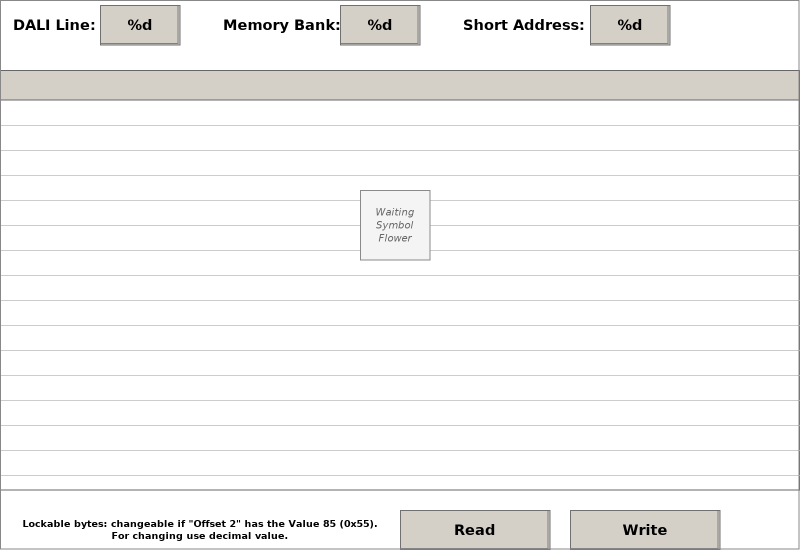
VISUALIZATION Visu_Part102MemoryBank  // 800x550
    Table (0,70 800x420), data array: DALI_Commissioning.fbPart102MemoryPages.aMemoryBank
        p1137915858: DALI_Commissioning.fbPart102MemoryPages.nOffset
        p3854506369: DALI_Commissioning.fbPart102MemoryPages.aMemoryBank[INDEX].sOffset
        p1892666644: DALI_Commissioning.fbPart102MemoryPages.aMemoryBank[INDEX].sName
        p338671338: DALI_Commissioning.fbPart102MemoryPages.aMemoryBank[INDEX].nValueDec
        p2170511999: DALI_Commissioning.fbPart102MemoryPages.aMemoryBank[INDEX].nValueHex
        p1755163831: Value Dec
        p4092479075: Value Hex
        Columns.Column.[0].Template: DALI_Commissioning.fbPart102MemoryPages.aNoValue[INDEX]
        Columns.Column.[1].Template: DALI_Commissioning.fbPart102MemoryPages.aNoValue[INDEX]
        Columns.Column.[2].Template: DALI_Commissioning.fbPart102MemoryPages.aNoValue[INDEX]; OnMouseClick: write the text variable via Default, min 0, max 255, title "Lockable variable decimal"
        Columns.Column.[3].Template: DALI_Commissioning.fbPart102MemoryPages.aNoValue[INDEX]; OnMouseClick: write the text variable via Default, title "Lockable variable hexadecimal"
    Button (400,510 150x40), "Read"
        OnMouseClick: execute { DALI_Commissioning.fbPart102MemoryPages.bRead := TRUE; }
    Button (570,510 150x40), "Write"
        OnMouseClick: execute { DALI_Commissioning.fbPart102MemoryPages.bWrite := TRUE; }
    Textfield (15,510 370x40), "Lockable bytes: changeable if "Offset 2" has the Value 85 (0x55). For changing use decimal value."
    WaitingSymbolFlower (360,190 70x70), invisible if: DALI_Commissioning.fbPart102MemoryPages.bHideWaitSymbol
    Textfield (460,5 130x40), "Short Address:"
    Button (590,5 80x40), "%d", text variable: DALI_Commissioning.fbPart102MemoryPages.nAddress
        OnMouseClick: write the text variable via Default, min 0, max 63, title "Insert Short Address"
    Textfield (220,5 120x40), "Memory Bank:"
    Button (340,5 80x40), "%d", text variable: DALI_Commissioning.fbPart102MemoryPages.nMemoryBank
        OnMouseClick: write the text variable via Default, min 0, max 255, title "Insert Memory Bank"
    Group (10,5 170x40)
        Textfield (0,0 110x40), "DALI Line:"
        Button (90,0 80x40), "%d", text variable: GVL_Internal.nDALILine
            OnMouseClick: write the text variable via Default, min 1, max 10, title "Choose line"
END_VISUALIZATION

(* stored: Version 1.1.0.1
   Visu Visu_Part102MemoryBank: Id {e33c44f6-d127-4b31-8006-ff2c4946b58f} *)
